FUNCTION_BLOCK NormallyClosePushButton IMPLEMENTS I_PushButton

VAR
	Input	AT %I* : BOOL; 
END_VAR

PROPERTY IsPressed : BOOL
GET
IsPressed := NOT Input;
END_GET
END_PROPERTY

PROPERTY IsReleased : BOOL
GET
IsReleased := NOT IsPressed;
END_GET
END_PROPERTY

END_FUNCTION_BLOCK

(* stored: Version 1.1.0.1, ProductVersion 3.1.4024.12
   POU NormallyClosePushButton: Id {dcfaa6f5-d5f6-4649-91bf-afd92debe649}, SpecialFunc None
   Property IsPressed: Id {2046154d-0544-4cbc-b41e-388a502d3ce4}
   Get Get: Id {49ef60e8-08f1-4091-b951-096e66c82f21}
   Property IsReleased: Id {a73def30-cdd2-4a57-8260-2132758c87f5}
   Get Get: Id {4b9d5916-9566-4ef5-a519-255dc0a85d79} *)
